FUNCTION_BLOCK SS3_ifb_Bunker (* Basic FB with empty ECC *)
  (* Standard: 61499-2 *)
  (* Version 1.0, 2021-08-03, AK121668 *)
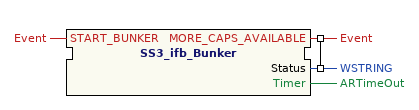
  EVENT_INPUT
    START_BUNKER; (* start feeding bunker *)
  END_EVENT
  EVENT_OUTPUT
    MORE_CAPS_AVAILABLE WITH Status; (* feeding is DONE *)
  END_EVENT
  VAR_OUTPUT
    Status : WSTRING; (* Current Status of Bunker *)
  END_VAR
  PLUGS
    Timer : ARTimeOut;
  END_PLUGS
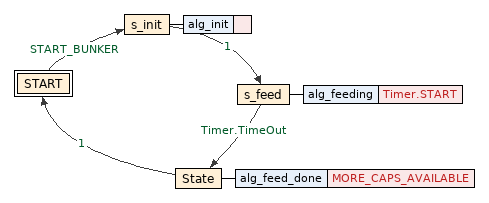
  EC_STATES
    START; (* Initial State *)
    s_feed : alg_feeding -> Timer.START;
    State : alg_feed_done -> MORE_CAPS_AVAILABLE;
    s_init : alg_init;
  END_STATES
  EC_TRANSITIONS
    s_feed TO State := Timer.TimeOut;
    State TO START := 1;
    START TO s_init := START_BUNKER;
    s_init TO s_feed := 1;
  END_TRANSITIONS
  ALGORITHM alg_init IN ST:
Timer.DT := T#5s;
Status := WSTRING#"init mode";
  END_ALGORITHM
  ALGORITHM alg_feeding IN ST:
Status := WSTRING#"feeding now";
  END_ALGORITHM
  ALGORITHM alg_feed_done IN ST:
Status := WSTRING#"feeding Done";
  END_ALGORITHM
  ALGORITHM alg_no_cap_alarm IN ST:
Status := WSTRING#"Caps not available";
  END_ALGORITHM
END_FUNCTION_BLOCK
